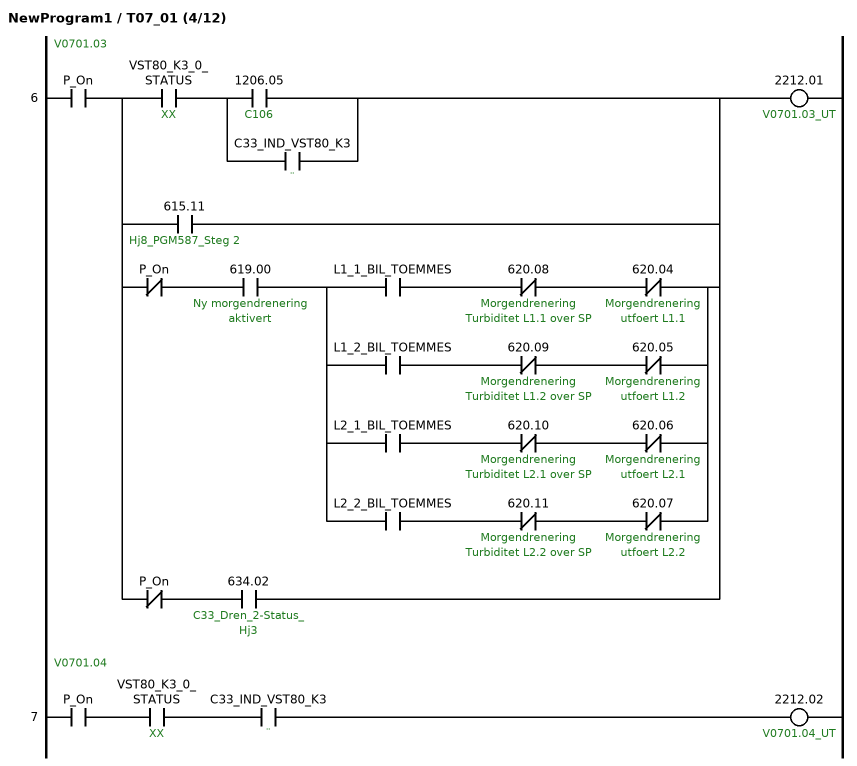
; [picture p960: NewProgram1 / T07_01, rungs 6-7]
; rung 6: V0701.03
LD P_On
LD VST80_K3_0_STATUS  ; XX
LD 1206.05  ; C106
OR C33_IND_VST80_K3  ; ¨
ANDLD
OR 615.11  ; Hj8_PGM587_Steg 2
LDNOT P_On
AND 619.00  ; Ny morgendrenering aktivert
LD L1_1_BIL_TOEMMES
ANDNOT 620.08  ; Morgendrenering Turbiditet L1.1 over SP
ANDNOT 620.04  ; Morgendrenering utfoert L1.1
LD L1_2_BIL_TOEMMES
ANDNOT 620.09  ; Morgendrenering Turbiditet L1.2 over SP
ANDNOT 620.05  ; Morgendrenering utfoert L1.2
ORLD
LD L2_1_BIL_TOEMMES
ANDNOT 620.10  ; Morgendrenering Turbiditet L2.1 over SP
ANDNOT 620.06  ; Morgendrenering utfoert L2.1
ORLD
LD L2_2_BIL_TOEMMES
ANDNOT 620.11  ; Morgendrenering Turbiditet L2.2 over SP
ANDNOT 620.07  ; Morgendrenering utfoert L2.2
ORLD
ANDLD
ORLD
LDNOT P_On
AND 634.02  ; C33_Dren_2-Status_Hj3
ORLD
ANDLD
OUT 2212.01  ; V0701.03_UT
; rung 7: V0701.04
LD P_On
AND VST80_K3_0_STATUS  ; XX
AND C33_IND_VST80_K3  ; ¨
OUT 2212.02  ; V0701.04_UT

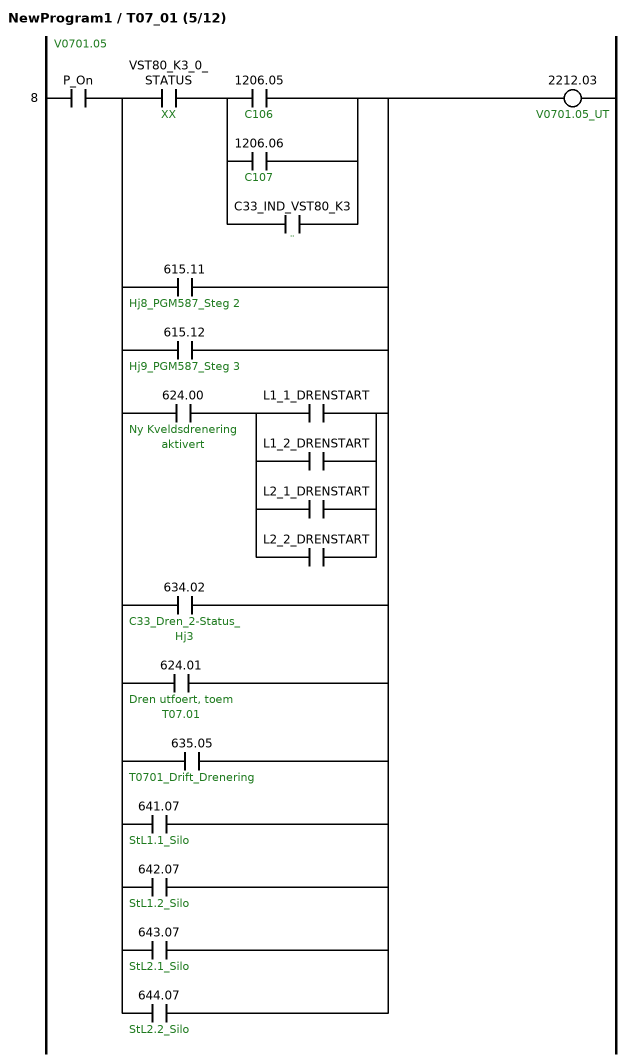
; rung 8: V0701.05
LD P_On
LD VST80_K3_0_STATUS  ; XX
LD 1206.05  ; C106
OR 1206.06  ; C107
OR C33_IND_VST80_K3  ; ¨
ANDLD
OR 615.11  ; Hj8_PGM587_Steg 2
OR 615.12  ; Hj9_PGM587_Steg 3
LD 624.00  ; Ny Kveldsdrenering aktivert
LD L1_1_DRENSTART
OR L1_2_DRENSTART
OR L2_1_DRENSTART
OR L2_2_DRENSTART
ANDLD
ORLD
OR 634.02  ; C33_Dren_2-Status_Hj3
OR 624.01  ; Dren utfoert, toem T07.01
OR 635.05  ; T0701_Drift_Drenering
OR 641.07  ; StL1.1_Silo
OR 642.07  ; StL1.2_Silo
OR 643.07  ; StL2.1_Silo
OR 644.07  ; StL2.2_Silo
ANDLD
OUT 2212.03  ; V0701.05_UT

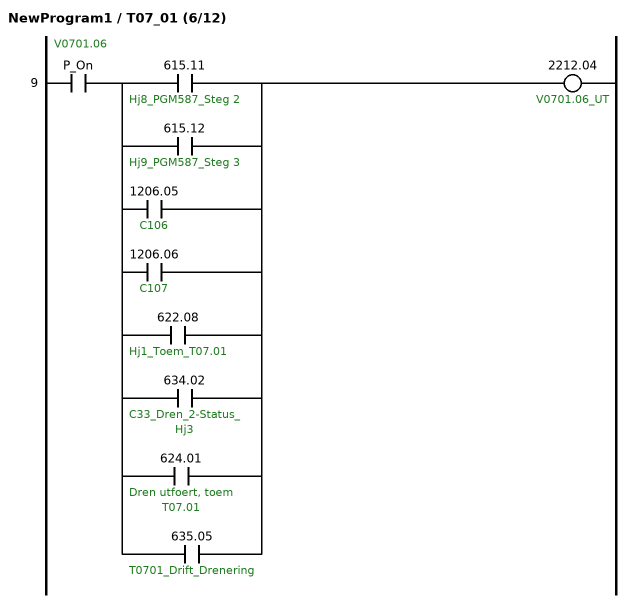
; rung 9: V0701.06
LD P_On
LD 615.11  ; Hj8_PGM587_Steg 2
OR 615.12  ; Hj9_PGM587_Steg 3
OR 1206.05  ; C106
OR 1206.06  ; C107
OR 622.08  ; Hj1_Toem_T07.01
OR 634.02  ; C33_Dren_2-Status_Hj3
OR 624.01  ; Dren utfoert, toem T07.01
OR 635.05  ; T0701_Drift_Drenering
ANDLD
OUT 2212.04  ; V0701.06_UT

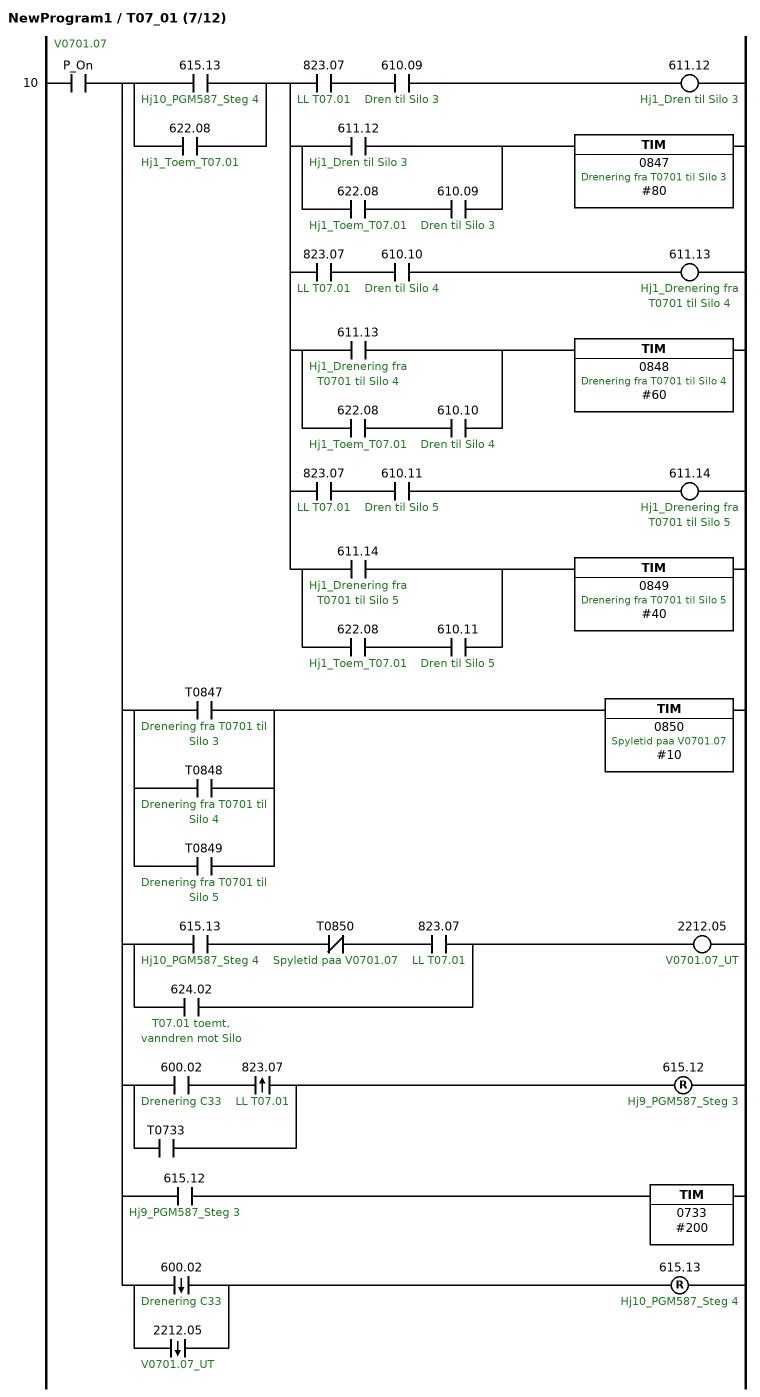
; rung 10: V0701.07
LD P_On
OUT TR0
LD 615.13  ; Hj10_PGM587_Steg 4
OR 622.08  ; Hj1_Toem_T07.01
ANDLD
OUT TR1
AND 823.07  ; LL T07.01
AND 610.09  ; Dren til Silo 3
OUT 611.12  ; Hj1_Dren til Silo 3
LD TR1
LD 611.12  ; Hj1_Dren til Silo 3
LD 622.08  ; Hj1_Toem_T07.01
AND 610.09  ; Dren til Silo 3
ORLD
ANDLD
TIM 0847 #80  ; Drenering fra T0701 til Silo 3
LD TR1
AND 823.07  ; LL T07.01
AND 610.10  ; Dren til Silo 4
OUT 611.13  ; Hj1_Drenering fra T0701 til Silo 4
LD TR1
LD 611.13  ; Hj1_Drenering fra T0701 til Silo 4
LD 622.08  ; Hj1_Toem_T07.01
AND 610.10  ; Dren til Silo 4
ORLD
ANDLD
TIM 0848 #60  ; Drenering fra T0701 til Silo 4
LD TR1
AND 823.07  ; LL T07.01
AND 610.11  ; Dren til Silo 5
OUT 611.14  ; Hj1_Drenering fra T0701 til Silo 5
LD TR1
LD 611.14  ; Hj1_Drenering fra T0701 til Silo 5
LD 622.08  ; Hj1_Toem_T07.01
AND 610.11  ; Dren til Silo 5
ORLD
ANDLD
TIM 0849 #40  ; Drenering fra T0701 til Silo 5
LD TR0
LD T0847  ; Drenering fra T0701 til Silo 3
OR T0848  ; Drenering fra T0701 til Silo 4
OR T0849  ; Drenering fra T0701 til Silo 5
ANDLD
TIM 0850 #10  ; Spyletid paa V0701.07
LD TR0
LD 615.13  ; Hj10_PGM587_Steg 4
ANDNOT T0850  ; Spyletid paa V0701.07
AND 823.07  ; LL T07.01
OR 624.02  ; T07.01 toemt, vanndren mot Silo
ANDLD
OUT 2212.05  ; V0701.07_UT
LD TR0
LD 600.02  ; Drenering C33
@AND 823.07  ; LL T07.01
OR T0733
ANDLD
RSET 615.12  ; Hj9_PGM587_Steg 3
LD TR0
AND 615.12  ; Hj9_PGM587_Steg 3
TIM 0733 #200
LD TR0
%LD 600.02  ; Drenering C33
%OR 2212.05  ; V0701.07_UT
ANDLD
RSET 615.13  ; Hj10_PGM587_Steg 4

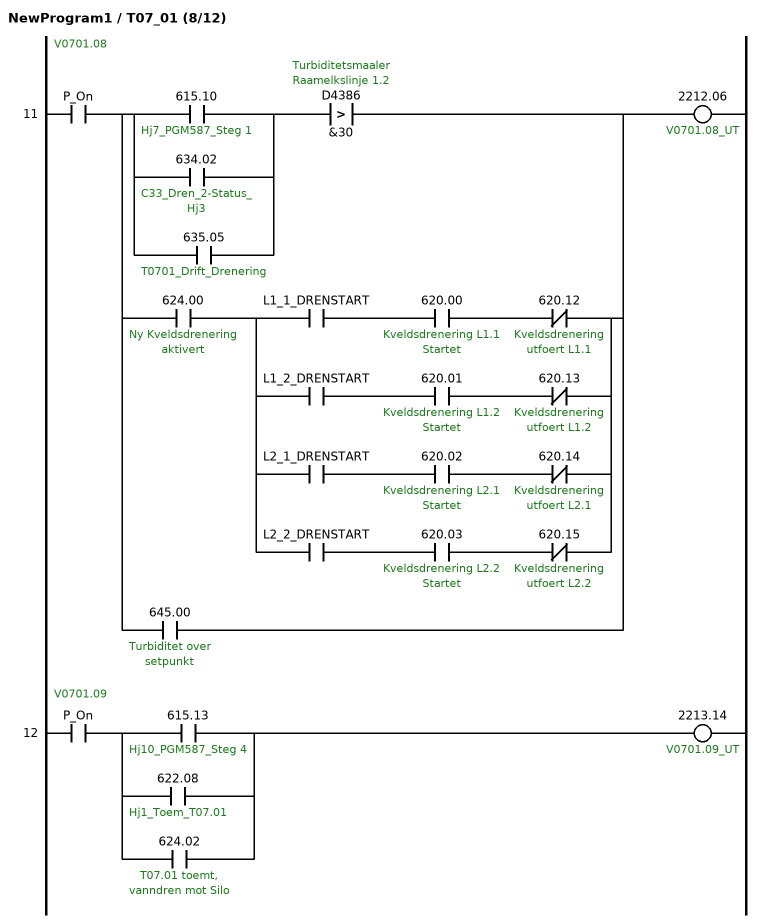
; rung 11: V0701.08
LD P_On
LD 615.10  ; Hj7_PGM587_Steg 1
OR 634.02  ; C33_Dren_2-Status_Hj3
OR 635.05  ; T0701_Drift_Drenering
AND>(320) D4386 &30  ; Turbiditetsmaaler Raamelkslinje 1.2
LD 624.00  ; Ny Kveldsdrenering aktivert
LD L1_1_DRENSTART
AND 620.00  ; Kveldsdrenering L1.1 Startet
ANDNOT 620.12  ; Kveldsdrenering utfoert L1.1
LD L1_2_DRENSTART
AND 620.01  ; Kveldsdrenering L1.2 Startet
ANDNOT 620.13  ; Kveldsdrenering utfoert L1.2
ORLD
LD L2_1_DRENSTART
AND 620.02  ; Kveldsdrenering L2.1 Startet
ANDNOT 620.14  ; Kveldsdrenering utfoert L2.1
ORLD
LD L2_2_DRENSTART
AND 620.03  ; Kveldsdrenering L2.2 Startet
ANDNOT 620.15  ; Kveldsdrenering utfoert L2.2
ORLD
ANDLD
ORLD
OR 645.00  ; Turbiditet over setpunkt
ANDLD
OUT 2212.06  ; V0701.08_UT
; rung 12: V0701.09
LD P_On
LD 615.13  ; Hj10_PGM587_Steg 4
OR 622.08  ; Hj1_Toem_T07.01
OR 624.02  ; T07.01 toemt, vanndren mot Silo
ANDLD
OUT 2213.14  ; V0701.09_UT

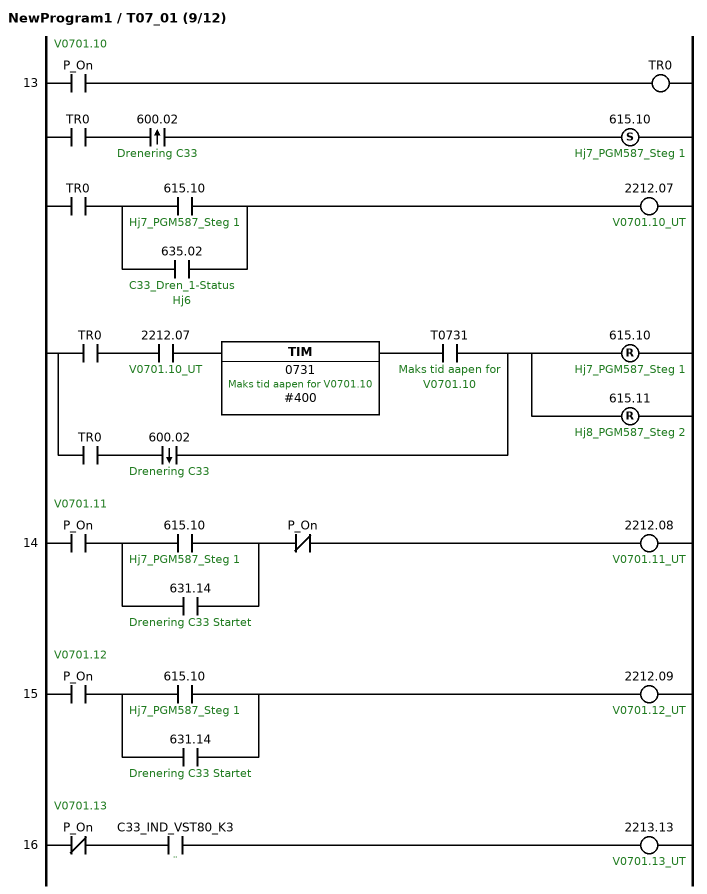
; rung 13: V0701.10
LD P_On
OUT TR0
@AND 600.02  ; Drenering C33
SET 615.10  ; Hj7_PGM587_Steg 1
LD TR0
LD 615.10  ; Hj7_PGM587_Steg 1
OR 635.02  ; C33_Dren_1-Status Hj6
ANDLD
OUT 2212.07  ; V0701.10_UT
LD TR0
AND 2212.07  ; V0701.10_UT
TIM 0731 #400  ; Maks tid aapen for V0701.10
AND T0731  ; Maks tid aapen for V0701.10
LD TR0
%AND 600.02  ; Drenering C33
ORLD
RSET 615.10  ; Hj7_PGM587_Steg 1
RSET 615.11  ; Hj8_PGM587_Steg 2
; rung 14: V0701.11
LD P_On
LD 615.10  ; Hj7_PGM587_Steg 1
OR 631.14  ; Drenering C33 Startet
ANDLD
ANDNOT P_On
OUT 2212.08  ; V0701.11_UT
; rung 15: V0701.12
LD P_On
LD 615.10  ; Hj7_PGM587_Steg 1
OR 631.14  ; Drenering C33 Startet
ANDLD
OUT 2212.09  ; V0701.12_UT
; rung 16: V0701.13
LDNOT P_On
AND C33_IND_VST80_K3  ; ¨
OUT 2213.13  ; V0701.13_UT

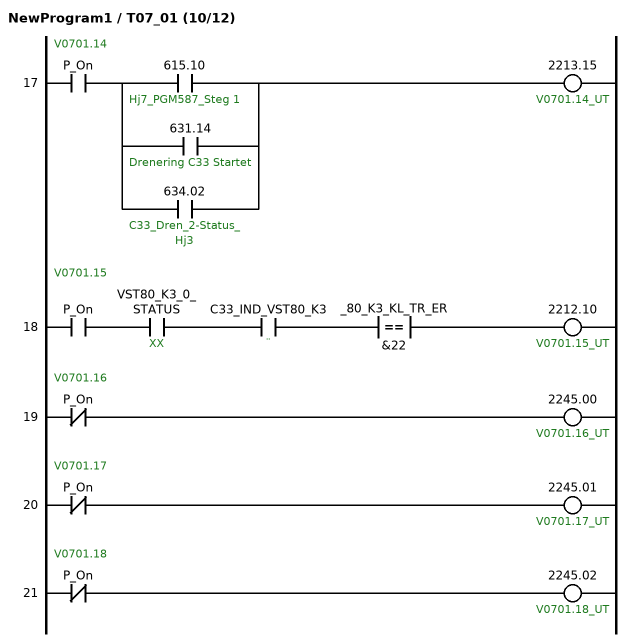
; rung 17: V0701.14
LD P_On
LD 615.10  ; Hj7_PGM587_Steg 1
OR 631.14  ; Drenering C33 Startet
OR 634.02  ; C33_Dren_2-Status_Hj3
ANDLD
OUT 2213.15  ; V0701.14_UT
; rung 18: V0701.15
LD P_On
AND VST80_K3_0_STATUS  ; XX
AND C33_IND_VST80_K3  ; ¨
AND=(300) _80_K3_KL_TR_ER &22
OUT 2212.10  ; V0701.15_UT
; rung 19: V0701.16
LDNOT P_On
OUT 2245.00  ; V0701.16_UT
; rung 20: V0701.17
LDNOT P_On
OUT 2245.01  ; V0701.17_UT
; rung 21: V0701.18
LDNOT P_On
OUT 2245.02  ; V0701.18_UT

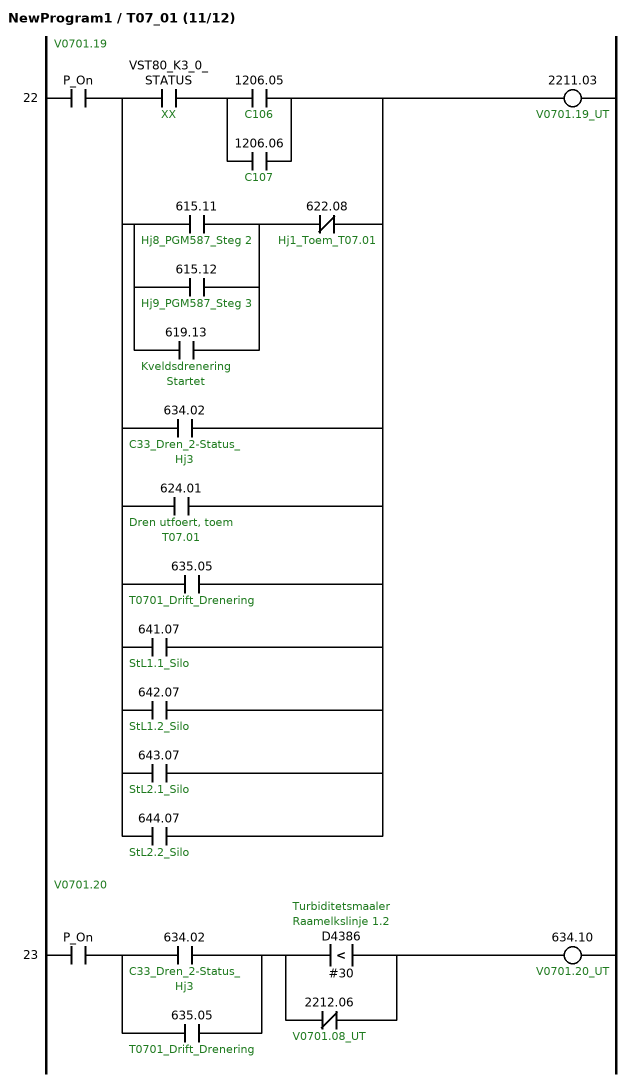
; rung 22: V0701.19
LD P_On
LD VST80_K3_0_STATUS  ; XX
LD 1206.05  ; C106
OR 1206.06  ; C107
ANDLD
LD 615.11  ; Hj8_PGM587_Steg 2
OR 615.12  ; Hj9_PGM587_Steg 3
OR 619.13  ; Kveldsdrenering Startet
ANDNOT 622.08  ; Hj1_Toem_T07.01
ORLD
OR 634.02  ; C33_Dren_2-Status_Hj3
OR 624.01  ; Dren utfoert, toem T07.01
OR 635.05  ; T0701_Drift_Drenering
OR 641.07  ; StL1.1_Silo
OR 642.07  ; StL1.2_Silo
OR 643.07  ; StL2.1_Silo
OR 644.07  ; StL2.2_Silo
ANDLD
OUT 2211.03  ; V0701.19_UT
; rung 23: V0701.20
LD P_On
LD 634.02  ; C33_Dren_2-Status_Hj3
OR 635.05  ; T0701_Drift_Drenering
ANDLD
LD<(310) D4386 #30  ; Turbiditetsmaaler Raamelkslinje 1.2
ORNOT 2212.06  ; V0701.08_UT
ANDLD
OUT 634.10  ; V0701.20_UT

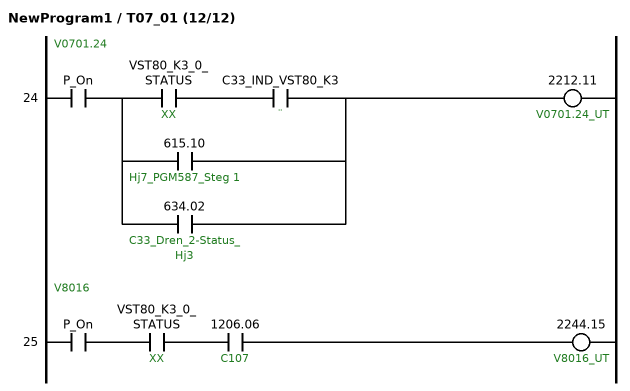
; rung 24: V0701.24
LD P_On
LD VST80_K3_0_STATUS  ; XX
AND C33_IND_VST80_K3  ; ¨
OR 615.10  ; Hj7_PGM587_Steg 1
OR 634.02  ; C33_Dren_2-Status_Hj3
ANDLD
OUT 2212.11  ; V0701.24_UT
; rung 25: V8016
LD P_On
AND VST80_K3_0_STATUS  ; XX
AND 1206.06  ; C107
OUT 2244.15  ; V8016_UT

### Section T07_02

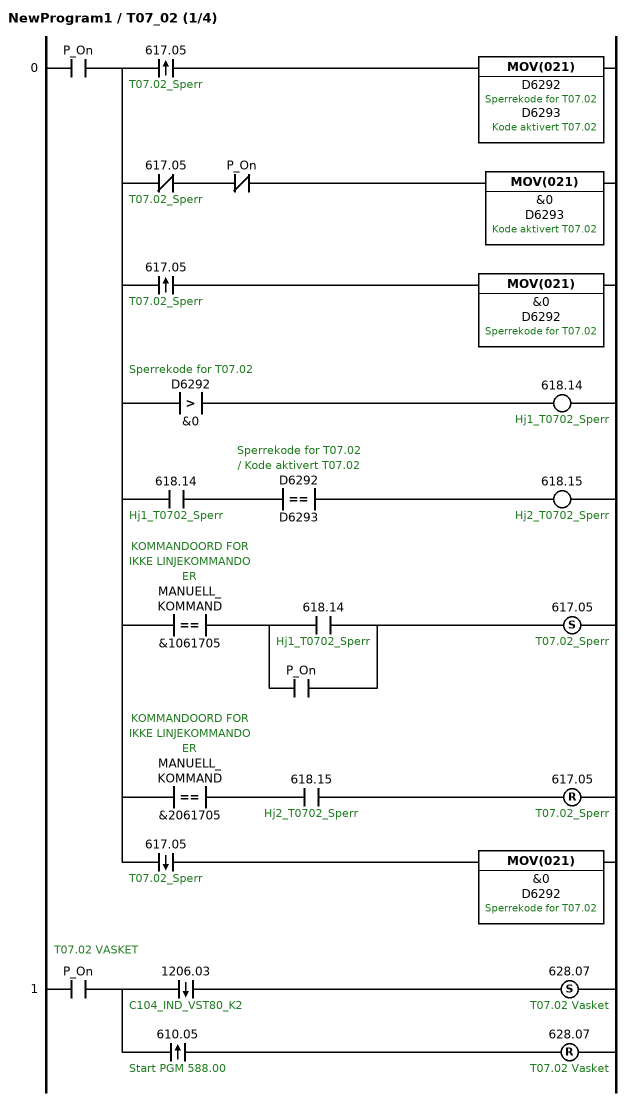
; rung 0
LD P_On
OUT TR0
@AND 617.05  ; T07.02_Sperr
MOV(021) D6292 D6293  ; Sperrekode for T07.02, Kode aktivert T07.02
LD TR0
ANDNOT 617.05  ; T07.02_Sperr
ANDNOT P_On
MOV(021) &0 D6293  ; Kode aktivert T07.02
LD TR0
@AND 617.05  ; T07.02_Sperr
MOV(021) &0 D6292  ; Sperrekode for T07.02
LD TR0
AND>(320) D6292 &0  ; Sperrekode for T07.02
OUT 618.14  ; Hj1_T0702_Sperr
LD TR0
AND 618.14  ; Hj1_T0702_Sperr
AND=(300) D6292 D6293  ; Sperrekode for T07.02, Kode aktivert T07.02
OUT 618.15  ; Hj2_T0702_Sperr
LD TR0
AND=L(301) MANUELL_KOMMAND &1061705  ; KOMMANDOORD FOR IKKE LINJEKOMMANDOER
LD 618.14  ; Hj1_T0702_Sperr
OR P_On
ANDLD
SET 617.05  ; T07.02_Sperr
LD TR0
AND=L(301) MANUELL_KOMMAND &2061705  ; KOMMANDOORD FOR IKKE LINJEKOMMANDOER
AND 618.15  ; Hj2_T0702_Sperr
RSET 617.05  ; T07.02_Sperr
LD TR0
%AND 617.05  ; T07.02_Sperr
MOV(021) &0 D6292  ; Sperrekode for T07.02
; rung 1: T07.02 VASKET
LD P_On
OUT TR0
%AND 1206.03  ; C104_IND_VST80_K2
SET 628.07  ; T07.02 Vasket
LD TR0
@AND 610.05  ; Start PGM 588.00
RSET 628.07  ; T07.02 Vasket

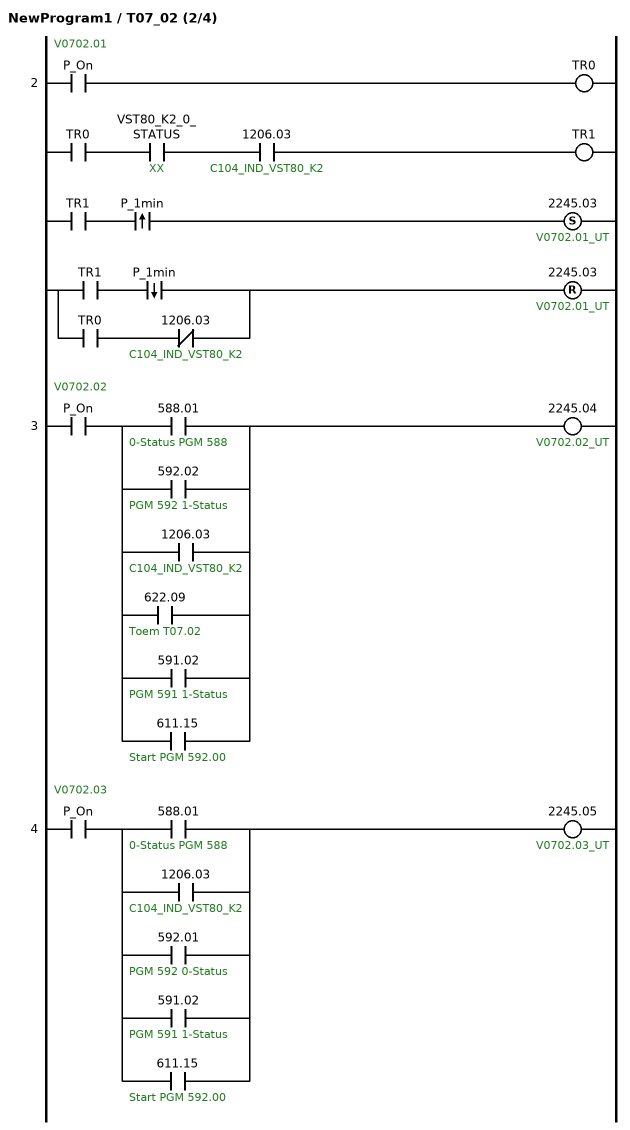
; rung 2: V0702.01
LD P_On
OUT TR0
AND VST80_K2_0_STATUS  ; XX
AND 1206.03  ; C104_IND_VST80_K2
OUT TR1
@AND P_1min
SET 2245.03  ; V0702.01_UT
LD TR1
%AND P_1min
LD TR0
ANDNOT 1206.03  ; C104_IND_VST80_K2
ORLD
RSET 2245.03  ; V0702.01_UT
; rung 3: V0702.02
LD P_On
LD 588.01  ; 0-Status PGM 588
OR 592.02  ; PGM 592 1-Status
OR 1206.03  ; C104_IND_VST80_K2
OR 622.09  ; Toem T07.02
OR 591.02  ; PGM 591 1-Status
OR 611.15  ; Start PGM 592.00
ANDLD
OUT 2245.04  ; V0702.02_UT
; rung 4: V0702.03
LD P_On
LD 588.01  ; 0-Status PGM 588
OR 1206.03  ; C104_IND_VST80_K2
OR 592.01  ; PGM 592 0-Status
OR 591.02  ; PGM 591 1-Status
OR 611.15  ; Start PGM 592.00
ANDLD
OUT 2245.05  ; V0702.03_UT

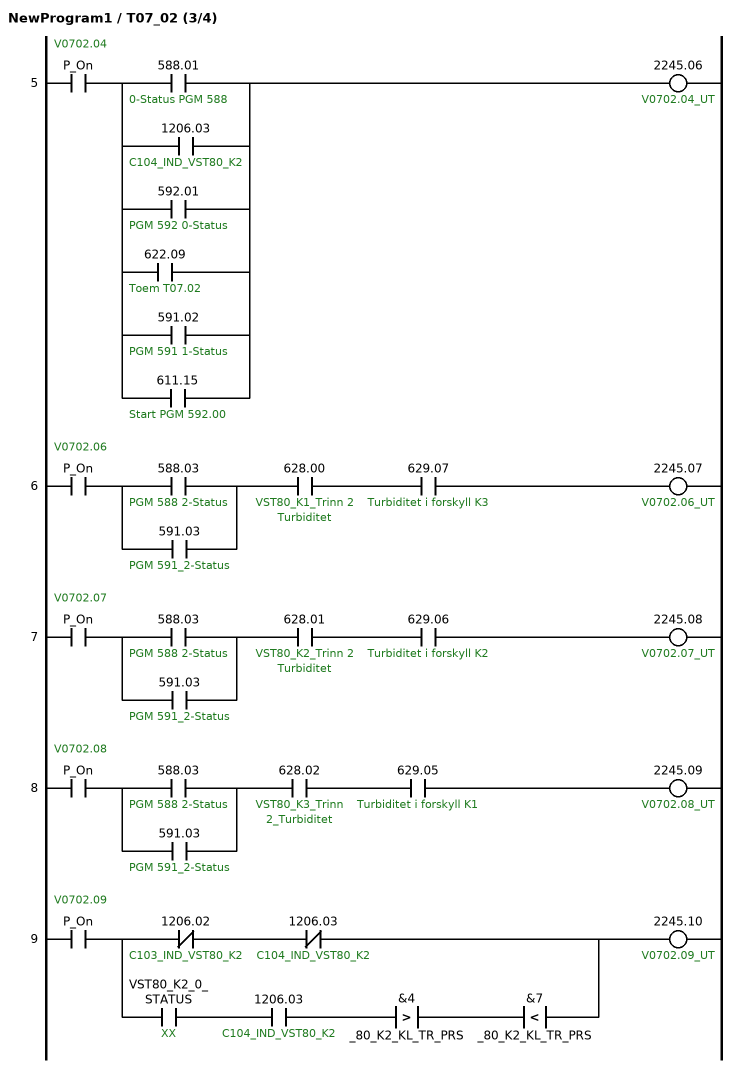
; rung 5: V0702.04
LD P_On
LD 588.01  ; 0-Status PGM 588
OR 1206.03  ; C104_IND_VST80_K2
OR 592.01  ; PGM 592 0-Status
OR 622.09  ; Toem T07.02
OR 591.02  ; PGM 591 1-Status
OR 611.15  ; Start PGM 592.00
ANDLD
OUT 2245.06  ; V0702.04_UT
; rung 6: V0702.06
LD P_On
LD 588.03  ; PGM 588 2-Status
OR 591.03  ; PGM 591_2-Status
ANDLD
AND 628.00  ; VST80_K1_Trinn 2 Turbiditet
AND 629.07  ; Turbiditet i forskyll K3
OUT 2245.07  ; V0702.06_UT
; rung 7: V0702.07
LD P_On
LD 588.03  ; PGM 588 2-Status
OR 591.03  ; PGM 591_2-Status
ANDLD
AND 628.01  ; VST80_K2_Trinn 2 Turbiditet
AND 629.06  ; Turbiditet i forskyll K2
OUT 2245.08  ; V0702.07_UT
; rung 8: V0702.08
LD P_On
LD 588.03  ; PGM 588 2-Status
OR 591.03  ; PGM 591_2-Status
ANDLD
AND 628.02  ; VST80_K3_Trinn 2_Turbiditet
AND 629.05  ; Turbiditet i forskyll K1
OUT 2245.09  ; V0702.08_UT
; rung 9: V0702.09
LD P_On
LDNOT 1206.02  ; C103_IND_VST80_K2
ANDNOT 1206.03  ; C104_IND_VST80_K2
LD VST80_K2_0_STATUS  ; XX
AND 1206.03  ; C104_IND_VST80_K2
AND>(320) &4 _80_K2_KL_TR_PRS
AND<(310) &7 _80_K2_KL_TR_PRS
ORLD
ANDLD
OUT 2245.10  ; V0702.09_UT

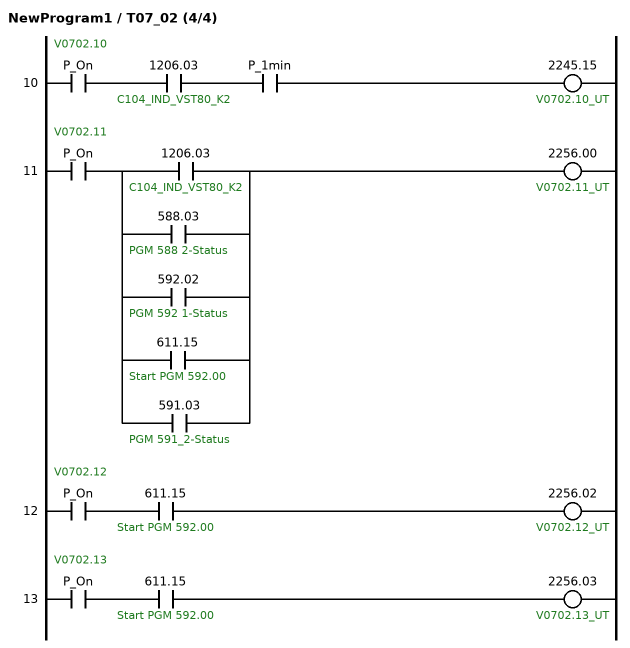
; rung 10: V0702.10
LD P_On
AND 1206.03  ; C104_IND_VST80_K2
AND P_1min
OUT 2245.15  ; V0702.10_UT
; rung 11: V0702.11
LD P_On
LD 1206.03  ; C104_IND_VST80_K2
OR 588.03  ; PGM 588 2-Status
OR 592.02  ; PGM 592 1-Status
OR 611.15  ; Start PGM 592.00
OR 591.03  ; PGM 591_2-Status
ANDLD
OUT 2256.00  ; V0702.11_UT
; rung 12: V0702.12
LD P_On
AND 611.15  ; Start PGM 592.00
OUT 2256.02  ; V0702.12_UT
; rung 13: V0702.13
LD P_On
AND 611.15  ; Start PGM 592.00
OUT 2256.03  ; V0702.13_UT

### Section T24_TEMP_NIVÅ

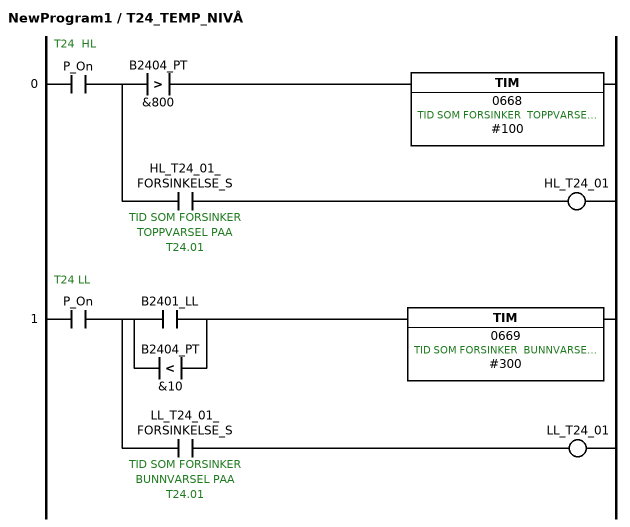
; rung 0: T24  HL
LD P_On
OUT TR0
AND>(320) B2404_PT &800
TIM 0668 #100  ; TID SOM FORSINKER  TOPPVARSEL PAA T24.01
LD TR0
AND HL_T24_01_FORSINKELSE_S  ; TID SOM FORSINKER  TOPPVARSEL PAA T24.01
OUT HL_T24_01
; rung 1: T24 LL
LD P_On
OUT TR0
LD B2401_LL
OR<(310) B2404_PT &10
ANDLD
TIM 0669 #300  ; TID SOM FORSINKER  BUNNVARSEL PAA T24.01
LD TR0
AND LL_T24_01_FORSINKELSE_S  ; TID SOM FORSINKER  BUNNVARSEL PAA T24.01
OUT LL_T24_01

### Section T24_STATUS

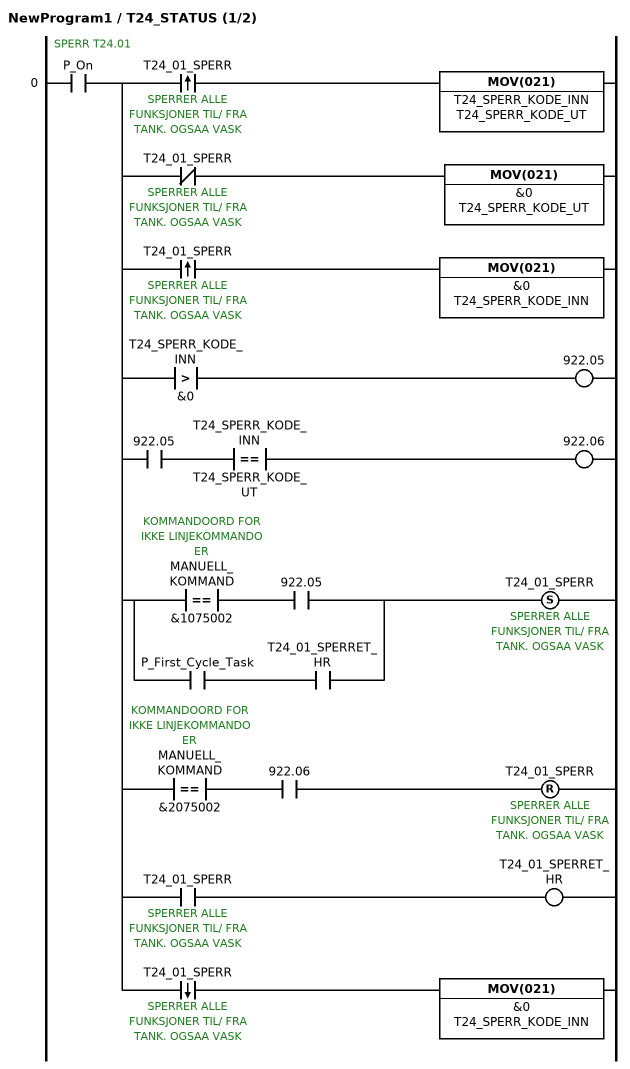
; rung 0: SPERR T24.01
LD P_On
OUT TR0
@AND T24_01_SPERR  ; SPERRER ALLE FUNKSJONER TIL/ FRA TANK. OGSAA VASK
MOV(021) T24_SPERR_KODE_INN T24_SPERR_KODE_UT
LD TR0
ANDNOT T24_01_SPERR  ; SPERRER ALLE FUNKSJONER TIL/ FRA TANK. OGSAA VASK
MOV(021) &0 T24_SPERR_KODE_UT
LD TR0
@AND T24_01_SPERR  ; SPERRER ALLE FUNKSJONER TIL/ FRA TANK. OGSAA VASK
MOV(021) &0 T24_SPERR_KODE_INN
LD TR0
AND>(320) T24_SPERR_KODE_INN &0
OUT 922.05
LD TR0
AND 922.05
AND=(300) T24_SPERR_KODE_INN T24_SPERR_KODE_UT
OUT 922.06
LD TR0
LD=L(301) MANUELL_KOMMAND &1075002  ; KOMMANDOORD FOR IKKE LINJEKOMMANDOER
AND 922.05
LD P_First_Cycle_Task
AND T24_01_SPERRET_HR
ORLD
ANDLD
SET T24_01_SPERR  ; SPERRER ALLE FUNKSJONER TIL/ FRA TANK. OGSAA VASK
LD TR0
AND=L(301) MANUELL_KOMMAND &2075002  ; KOMMANDOORD FOR IKKE LINJEKOMMANDOER
AND 922.06
RSET T24_01_SPERR  ; SPERRER ALLE FUNKSJONER TIL/ FRA TANK. OGSAA VASK
LD TR0
AND T24_01_SPERR  ; SPERRER ALLE FUNKSJONER TIL/ FRA TANK. OGSAA VASK
OUT T24_01_SPERRET_HR
LD TR0
%AND T24_01_SPERR  ; SPERRER ALLE FUNKSJONER TIL/ FRA TANK. OGSAA VASK
MOV(021) &0 T24_SPERR_KODE_INN

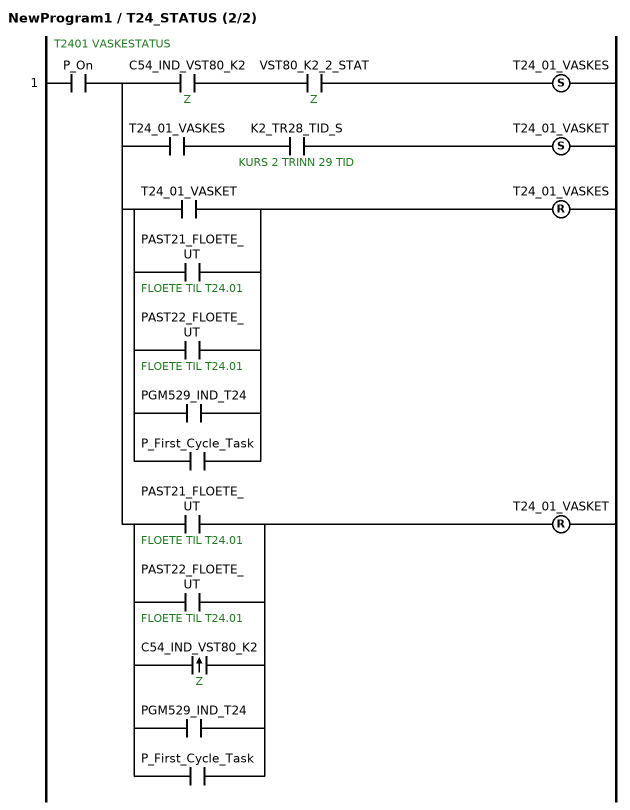
; rung 1: T2401 VASKESTATUS
LD P_On
OUT TR0
AND C54_IND_VST80_K2  ; Z
AND VST80_K2_2_STAT  ; Z
SET T24_01_VASKES
LD TR0
AND T24_01_VASKES
AND K2_TR28_TID_S  ; KURS 2 TRINN 29 TID
SET T24_01_VASKET
LD TR0
LD T24_01_VASKET
OR PAST21_FLOETE_UT  ; FLOETE TIL T24.01
OR PAST22_FLOETE_UT  ; FLOETE TIL T24.01
OR PGM529_IND_T24
OR P_First_Cycle_Task
ANDLD
RSET T24_01_VASKES
LD TR0
LD PAST21_FLOETE_UT  ; FLOETE TIL T24.01
OR PAST22_FLOETE_UT  ; FLOETE TIL T24.01
@OR C54_IND_VST80_K2  ; Z
OR PGM529_IND_T24
OR P_First_Cycle_Task
ANDLD
RSET T24_01_VASKET

### Section T24_VENTILER_OG_PUMPER

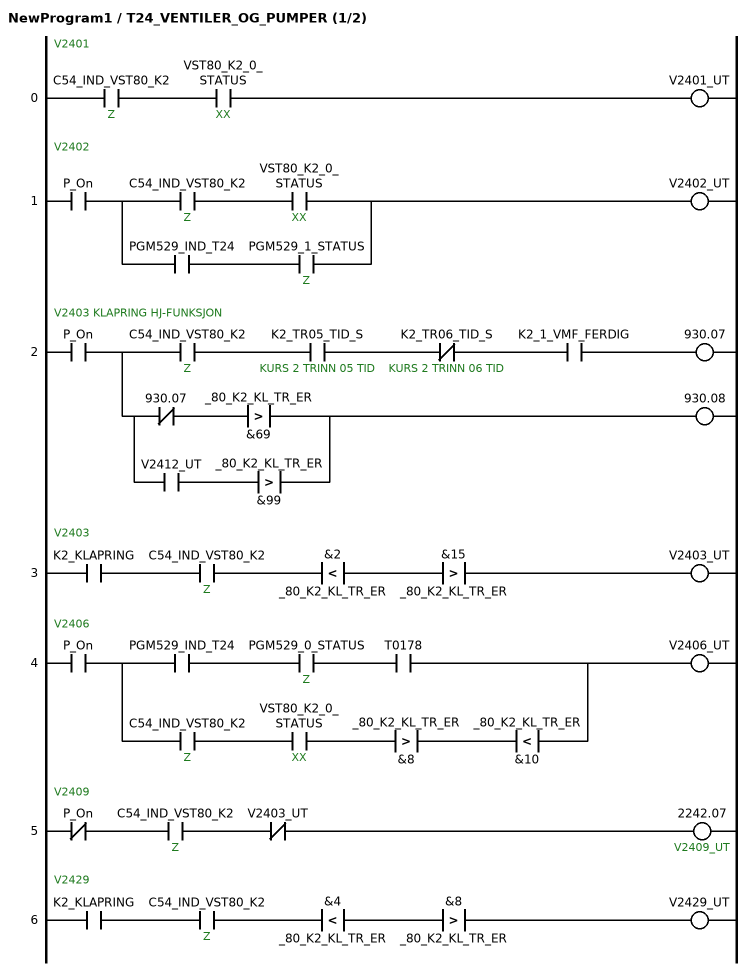
; rung 0: V2401
LD C54_IND_VST80_K2  ; Z
AND VST80_K2_0_STATUS  ; XX
OUT V2401_UT
; rung 1: V2402
LD P_On
LD C54_IND_VST80_K2  ; Z
AND VST80_K2_0_STATUS  ; XX
LD PGM529_IND_T24
AND PGM529_1_STATUS  ; Z
ORLD
ANDLD
OUT V2402_UT
; rung 2: V2403 KLAPRING HJ-FUNKSJON
LD P_On
OUT TR0
AND C54_IND_VST80_K2  ; Z
AND K2_TR05_TID_S  ; KURS 2 TRINN 05 TID
ANDNOT K2_TR06_TID_S  ; KURS 2 TRINN 06 TID
AND K2_1_VMF_FERDIG
OUT 930.07
LD TR0
LDNOT 930.07
AND>(320) _80_K2_KL_TR_ER &69
LD V2412_UT
AND>(320) _80_K2_KL_TR_ER &99
ORLD
ANDLD
OUT 930.08
; rung 3: V2403
LD K2_KLAPRING
AND C54_IND_VST80_K2  ; Z
AND<(310) &2 _80_K2_KL_TR_ER
AND>(320) &15 _80_K2_KL_TR_ER
OUT V2403_UT
; rung 4: V2406
LD P_On
LD PGM529_IND_T24
AND PGM529_0_STATUS  ; Z
AND T0178
LD C54_IND_VST80_K2  ; Z
AND VST80_K2_0_STATUS  ; XX
AND>(320) _80_K2_KL_TR_ER &8
AND<(310) _80_K2_KL_TR_ER &10
ORLD
ANDLD
OUT V2406_UT
; rung 5: V2409
LDNOT P_On
AND C54_IND_VST80_K2  ; Z
ANDNOT V2403_UT
OUT 2242.07  ; V2409_UT
; rung 6: V2429
LD K2_KLAPRING
AND C54_IND_VST80_K2  ; Z
AND<(310) &4 _80_K2_KL_TR_ER
AND>(320) &8 _80_K2_KL_TR_ER
OUT V2429_UT

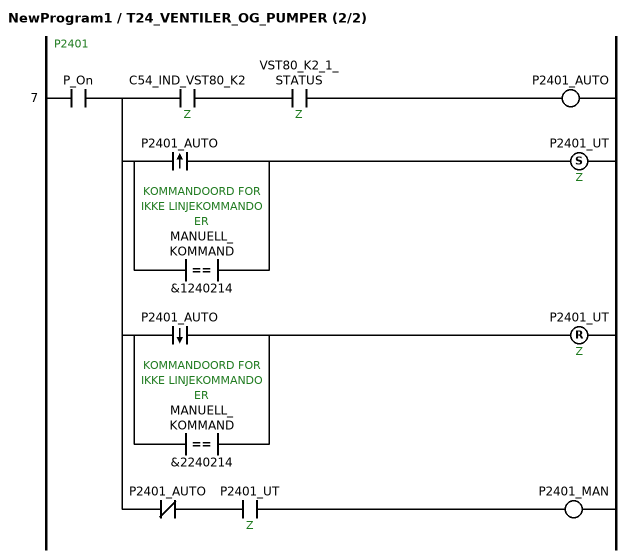
; rung 7: P2401
LD P_On
OUT TR0
AND C54_IND_VST80_K2  ; Z
AND VST80_K2_1_STATUS  ; Z
OUT P2401_AUTO
LD TR0
@LD P2401_AUTO
OR=L(301) MANUELL_KOMMAND &1240214  ; KOMMANDOORD FOR IKKE LINJEKOMMANDOER
ANDLD
SET P2401_UT  ; Z
LD TR0
%LD P2401_AUTO
OR=L(301) MANUELL_KOMMAND &2240214  ; KOMMANDOORD FOR IKKE LINJEKOMMANDOER
ANDLD
RSET P2401_UT  ; Z
LD TR0
ANDNOT P2401_AUTO
AND P2401_UT  ; Z
OUT P2401_MAN

### Section T27_01_SPERR

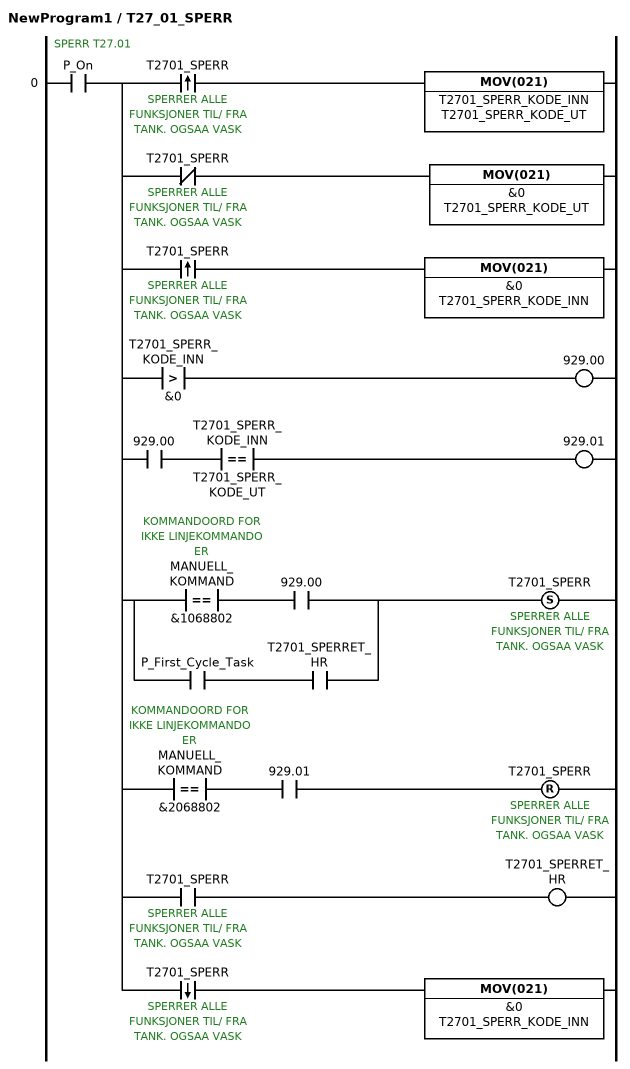
; rung 0: SPERR T27.01
LD P_On
OUT TR0
@AND T2701_SPERR  ; SPERRER ALLE FUNKSJONER TIL/ FRA TANK. OGSAA VASK
MOV(021) T2701_SPERR_KODE_INN T2701_SPERR_KODE_UT
LD TR0
ANDNOT T2701_SPERR  ; SPERRER ALLE FUNKSJONER TIL/ FRA TANK. OGSAA VASK
MOV(021) &0 T2701_SPERR_KODE_UT
LD TR0
@AND T2701_SPERR  ; SPERRER ALLE FUNKSJONER TIL/ FRA TANK. OGSAA VASK
MOV(021) &0 T2701_SPERR_KODE_INN
LD TR0
AND>(320) T2701_SPERR_KODE_INN &0
OUT 929.00
LD TR0
AND 929.00
AND=(300) T2701_SPERR_KODE_INN T2701_SPERR_KODE_UT
OUT 929.01
LD TR0
LD=L(301) MANUELL_KOMMAND &1068802  ; KOMMANDOORD FOR IKKE LINJEKOMMANDOER
AND 929.00
LD P_First_Cycle_Task
AND T2701_SPERRET_HR
ORLD
ANDLD
SET T2701_SPERR  ; SPERRER ALLE FUNKSJONER TIL/ FRA TANK. OGSAA VASK
LD TR0
AND=L(301) MANUELL_KOMMAND &2068802  ; KOMMANDOORD FOR IKKE LINJEKOMMANDOER
AND 929.01
RSET T2701_SPERR  ; SPERRER ALLE FUNKSJONER TIL/ FRA TANK. OGSAA VASK
LD TR0
AND T2701_SPERR  ; SPERRER ALLE FUNKSJONER TIL/ FRA TANK. OGSAA VASK
OUT T2701_SPERRET_HR
LD TR0
%AND T2701_SPERR  ; SPERRER ALLE FUNKSJONER TIL/ FRA TANK. OGSAA VASK
MOV(021) &0 T2701_SPERR_KODE_INN

### Section T27_01_NIVÅ

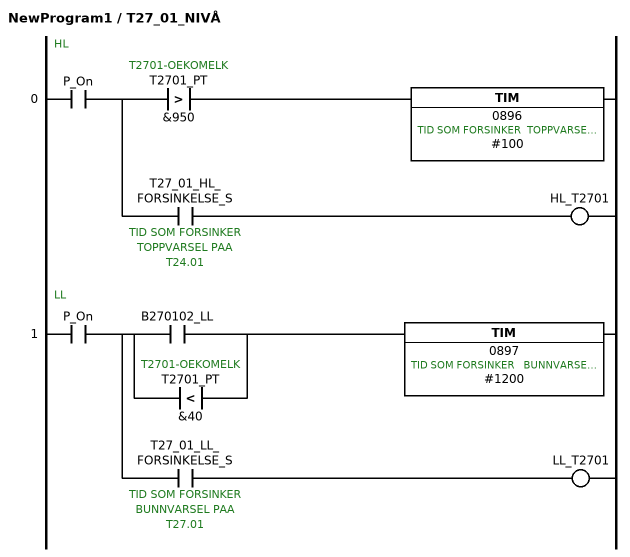
; rung 0: HL
LD P_On
OUT TR0
AND>(320) T2701_PT &950  ; T2701-OEKOMELK
TIM 0896 #100  ; TID SOM FORSINKER  TOPPVARSEL PAA T24.01
LD TR0
AND T27_01_HL_FORSINKELSE_S  ; TID SOM FORSINKER  TOPPVARSEL PAA T24.01
OUT HL_T2701
; rung 1: LL
LD P_On
OUT TR0
LD B270102_LL
OR<(310) T2701_PT &40  ; T2701-OEKOMELK
ANDLD
TIM 0897 #1200  ; TID SOM FORSINKER   BUNNVARSEL PAA T27.01
LD TR0
AND T27_01_LL_FORSINKELSE_S  ; TID SOM FORSINKER   BUNNVARSEL PAA T27.01
OUT LL_T2701

### Section OBJEKTER_T27_01_ØKO

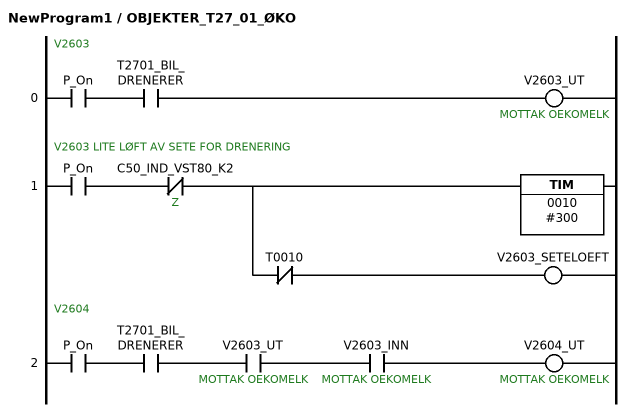
; rung 0: V2603
LD P_On
AND T2701_BIL_DRENERER
OUT V2603_UT  ; MOTTAK OEKOMELK
; rung 1: V2603 LITE LØFT AV SETE FOR DRENERING
LD P_On
ANDNOT C50_IND_VST80_K2  ; Z
TIM 0010 #300
ANDNOT T0010
OUT V2603_SETELOEFT
; rung 2: V2604
LD P_On
AND T2701_BIL_DRENERER
AND V2603_UT  ; MOTTAK OEKOMELK
AND V2603_INN  ; MOTTAK OEKOMELK
OUT V2604_UT  ; MOTTAK OEKOMELK

### Section T27_02_SPERR

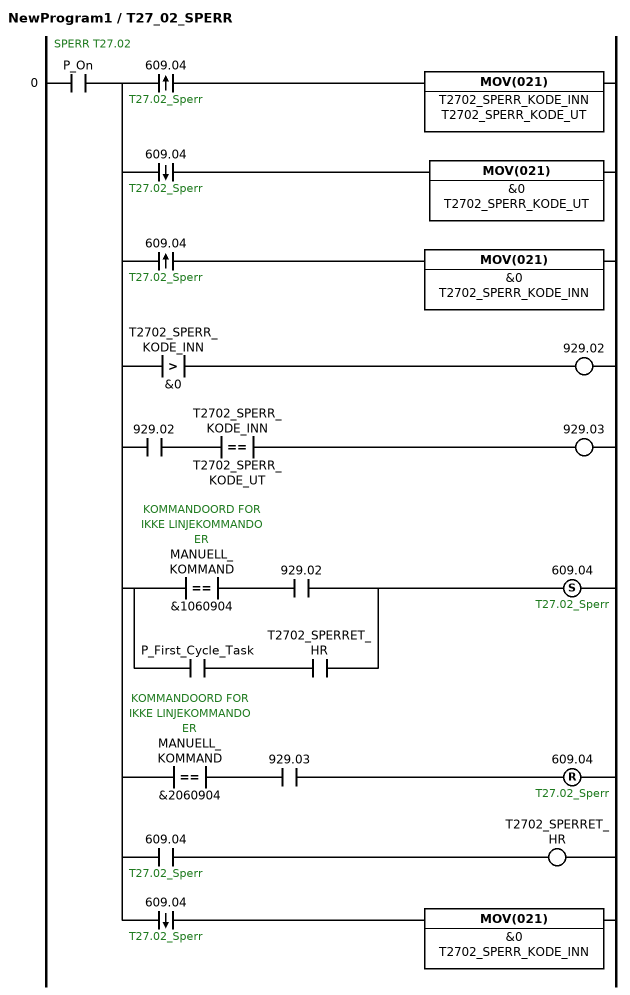
; rung 0: SPERR T27.02
LD P_On
OUT TR0
@AND 609.04  ; T27.02_Sperr
MOV(021) T2702_SPERR_KODE_INN T2702_SPERR_KODE_UT
LD TR0
%AND 609.04  ; T27.02_Sperr
MOV(021) &0 T2702_SPERR_KODE_UT
LD TR0
@AND 609.04  ; T27.02_Sperr
MOV(021) &0 T2702_SPERR_KODE_INN
LD TR0
AND>(320) T2702_SPERR_KODE_INN &0
OUT 929.02
LD TR0
AND 929.02
AND=(300) T2702_SPERR_KODE_INN T2702_SPERR_KODE_UT
OUT 929.03
LD TR0
LD=L(301) MANUELL_KOMMAND &1060904  ; KOMMANDOORD FOR IKKE LINJEKOMMANDOER
AND 929.02
LD P_First_Cycle_Task
AND T2702_SPERRET_HR
ORLD
ANDLD
SET 609.04  ; T27.02_Sperr
LD TR0
AND=L(301) MANUELL_KOMMAND &2060904  ; KOMMANDOORD FOR IKKE LINJEKOMMANDOER
AND 929.03
RSET 609.04  ; T27.02_Sperr
LD TR0
AND 609.04  ; T27.02_Sperr
OUT T2702_SPERRET_HR
LD TR0
%AND 609.04  ; T27.02_Sperr
MOV(021) &0 T2702_SPERR_KODE_INN

### Section T27_02_NIVÅ

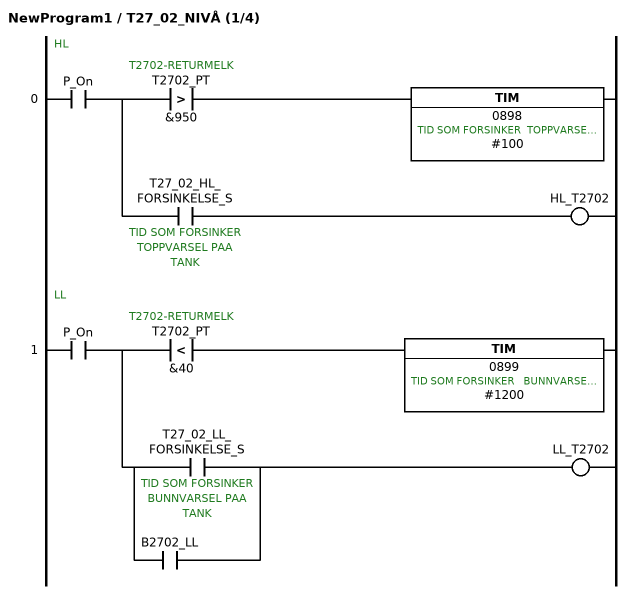
; rung 0: HL
LD P_On
OUT TR0
AND>(320) T2702_PT &950  ; T2702-RETURMELK
TIM 0898 #100  ; TID SOM FORSINKER  TOPPVARSEL PAA  TANK
LD TR0
AND T27_02_HL_FORSINKELSE_S  ; TID SOM FORSINKER  TOPPVARSEL PAA  TANK
OUT HL_T2702
; rung 1: LL
LD P_On
OUT TR0
AND<(310) T2702_PT &40  ; T2702-RETURMELK
TIM 0899 #1200  ; TID SOM FORSINKER   BUNNVARSEL PAA TANK
LD TR0
LD T27_02_LL_FORSINKELSE_S  ; TID SOM FORSINKER   BUNNVARSEL PAA TANK
OR B2702_LL
ANDLD
OUT LL_T2702

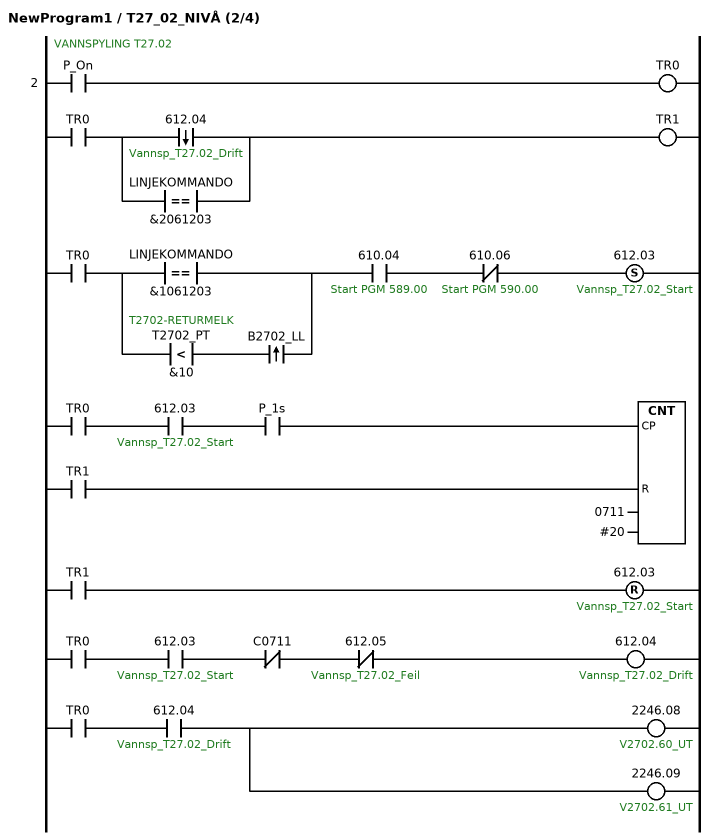
; rung 2: VANNSPYLING T27.02
LD P_On
OUT TR0
LD=L(301) LINJEKOMMANDO &1061203
LD<(310) T2702_PT &10  ; T2702-RETURMELK
@AND B2702_LL
ORLD
ANDLD
AND 610.04  ; Start PGM 589.00
ANDNOT 610.06  ; Start PGM 590.00
SET 612.03  ; Vannsp_T27.02_Start
LD TR0
AND 612.03  ; Vannsp_T27.02_Start
AND P_1s
LD TR0
%LD 612.04  ; Vannsp_T27.02_Drift
OR=L(301) LINJEKOMMANDO &2061203
ANDLD
OUT TR1
CNT 0711 #20
LD TR1
RSET 612.03  ; Vannsp_T27.02_Start
LD TR0
AND 612.03  ; Vannsp_T27.02_Start
ANDNOT C0711
ANDNOT 612.05  ; Vannsp_T27.02_Feil
OUT 612.04  ; Vannsp_T27.02_Drift
LD TR0
AND 612.04  ; Vannsp_T27.02_Drift
OUT 2246.08  ; V2702.60_UT
OUT 2246.09  ; V2702.61_UT

